{attribute 'qualified_only'}
VAR_GLOBAL
    Inputs AT %I* : ARRAY[0..7] OF BOOL;
    Outputs AT %Q* : ARRAY[0..7] OF BOOL;
END_VAR

(* stored: Version 1.1.0.1
   GVL gMANIPULATOR_IO: Id {906c05b5-124e-08ff-2366-1fb5554d91ef} *)
